// TIA Portal V17 export
FUNCTION "FC_MainControl" : Void   // FC, LAD
{ S7_Optimized_Access := 'TRUE' }
BEGIN

REGION Network 1: 风机运行联锁
   // 当风机运行按接通且风机故障反馈未动作时，驱动风机运行线圈
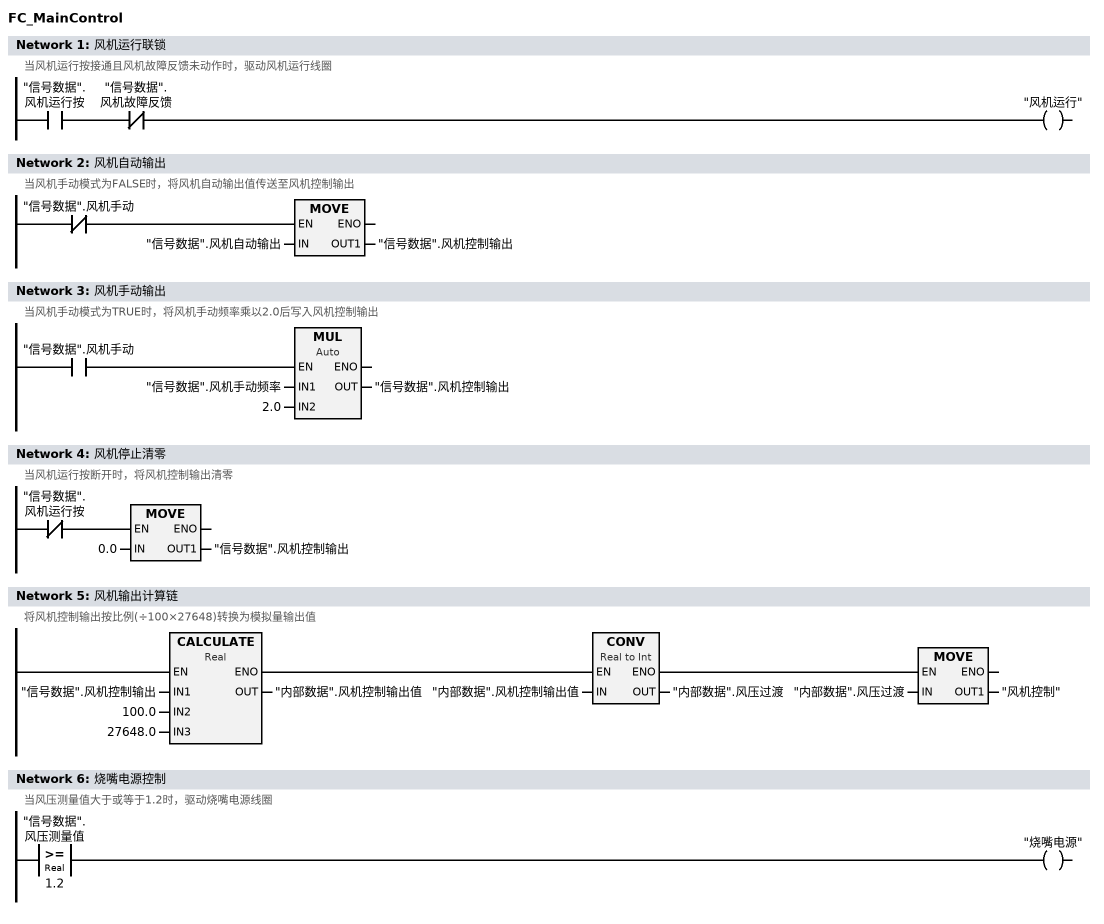
   RUNG wire#powerrail
      Contact( "信号数据".风机运行按 )
      I_Contact( "信号数据".风机故障反馈 )
      Coil( "风机运行" )
   END_RUNG
   // the same network as SCL:
   "风机运行" := "信号数据".风机运行按 AND NOT "信号数据".风机故障反馈;
END_REGION

REGION Network 2: 风机自动输出
   // 当风机手动模式为FALSE时，将风机自动输出值传送至风机控制输出
   RUNG wire#powerrail
      I_Contact( "信号数据".风机手动 )
      { S7_GenerateENO := "TRUE" } Move(in := "信号数据".风机自动输出, out1 => "信号数据".风机控制输出)
   END_RUNG
   // the same network as SCL:
   IF NOT "信号数据".风机手动 THEN "信号数据".风机控制输出 := "信号数据".风机自动输出; END_IF;
END_REGION

REGION Network 3: 风机手动输出
   // 当风机手动模式为TRUE时，将风机手动频率乘以2.0后写入风机控制输出
   RUNG wire#powerrail
      Contact( "信号数据".风机手动 )
      { S7_GenerateENO := "TRUE" } Mul(in1 := "信号数据".风机手动频率, in2 := 2.0, out => "信号数据".风机控制输出)
   END_RUNG
   // the same network as SCL:
   IF "信号数据".风机手动 THEN "信号数据".风机控制输出 := "信号数据".风机手动频率 * 2.0; END_IF;
END_REGION

REGION Network 4: 风机停止清零
   // 当风机运行按断开时，将风机控制输出清零
   RUNG wire#powerrail
      I_Contact( "信号数据".风机运行按 )
      { S7_GenerateENO := "TRUE" } Move(in := 0.0, out1 => "信号数据".风机控制输出)
   END_RUNG
   // the same network as SCL:
   IF NOT "信号数据".风机运行按 THEN "信号数据".风机控制输出 := 0.0; END_IF;
END_REGION

REGION Network 5: 风机输出计算链
   // 将风机控制输出按比例(÷100×27648)转换为模拟量输出值
   RUNG wire#powerrail
      { S7_Templates := "SrcType := Real"; S7_GenerateENO := "TRUE"; S7_Expression := "(IN1/IN2)*IN3" } Calculate(in1 := "信号数据".风机控制输出, in2 := 100.0, in3 := 27648.0, out => "内部数据".风机控制输出值)
      { S7_Templates := "[SrcType := Real, DestType := Int]"; S7_GenerateENO := "TRUE" } Convert(in := "内部数据".风机控制输出值, out => "内部数据".风压过渡)
      { S7_GenerateENO := "TRUE" } Move(in := "内部数据".风压过渡, out1 => "风机控制")
   END_RUNG
   // the same network as SCL:
   // ENO of a box is taken as its EN; it also drops when the box reports an error
   "内部数据".风机控制输出值 := ("信号数据".风机控制输出/100.0)*27648.0;
   "内部数据".风压过渡 := REAL_TO_INT("内部数据".风机控制输出值);
   "风机控制" := "内部数据".风压过渡;
END_REGION

REGION Network 6: 烧嘴电源控制
   // 当风压测量值大于或等于1.2时，驱动烧嘴电源线圈
   RUNG wire#powerrail
      { S7_Templates := "SrcType := Real" } GE_Contact(in1 := "信号数据".风压测量值, in2 := 1.2)
      Coil( "烧嘴电源" )
   END_RUNG
   // the same network as SCL:
   "烧嘴电源" := "信号数据".风压测量值 >= 1.2;
END_REGION
END_FUNCTION
